(* Logix 5000 project; controller Drives_Line1 1756-L72 rev 20.13; software revision 20.04; part 7 of 21 *)
(* tags used below, declared in another part *)
   Diamtest : BOOL;
   Diamtest_mm : REAL;
   Unwind_1_DiamCalcOn : BOOL;
   Unwinder_2_JEC : REAL;
   Unwinder_2_JLossCrvSpd : REAL[21];
   Unwinder_2_JMaterial : REAL;
   Unwinder_2_LossCrvTrq_Pct : REAL[21];
   Unwinder_2_MatMass : REAL;
   Unwinder_2_MatVolume : REAL;
   Unwinder_2_MaxMass : REAL;
   Unwinder_2_MaxVolume : REAL;
   Unwinder_2_PctPerN : REAL;
   Unwinder_2_RatedTrq : REAL;
   Unwinder_2_RPMPerMPS : REAL;
   zUnwind_2_MaxRate : REAL;
   zUnwind_2_TenRefRate : REAL;
   zUnwind_2_TenSpStall : REAL;
   zUnwind_2_TrqTrimLimMax_Pct : REAL;
   zUnwind_2_TrqTrimLimMin_Pct : REAL;
   zUnwinder_2_JGainQ1Q2 : REAL;
   zUnwinder_2_JGainQ3Q4 : REAL;
   zUnwinder_2_SpdReg_BWMax : REAL;
   zUnwinder_2_SpdReg_BWmin : REAL;
   Bridle_01 : UDT_Bridle_3M;
   EntryConfig : UDT_Config_Zone;
   EntryCtrl : UDT_Control_Zone;
   LineSetpoints : UDT_Setpoints_Line;
   Out_Feedbacks : UDT_Fdbks;
   Out_Status : UDT_Status;
   TestConfig_Unwinder_2 : UDT_Config_Unwinder;
   TestSp_Unwinder_2 : UDT_Setpoints_Unwinder;
   Unwinder_2 : UDT_Unwinder;
   Winder : UDT_Winder;
   zConfigFromMaster : BOOL;
   zPi : REAL;
(* P11_Unwinder_2, continued *)

ROUTINE R09_DiamCalc   (* function block diagram *)
   SHEET 1   // Distance/Angle Integration
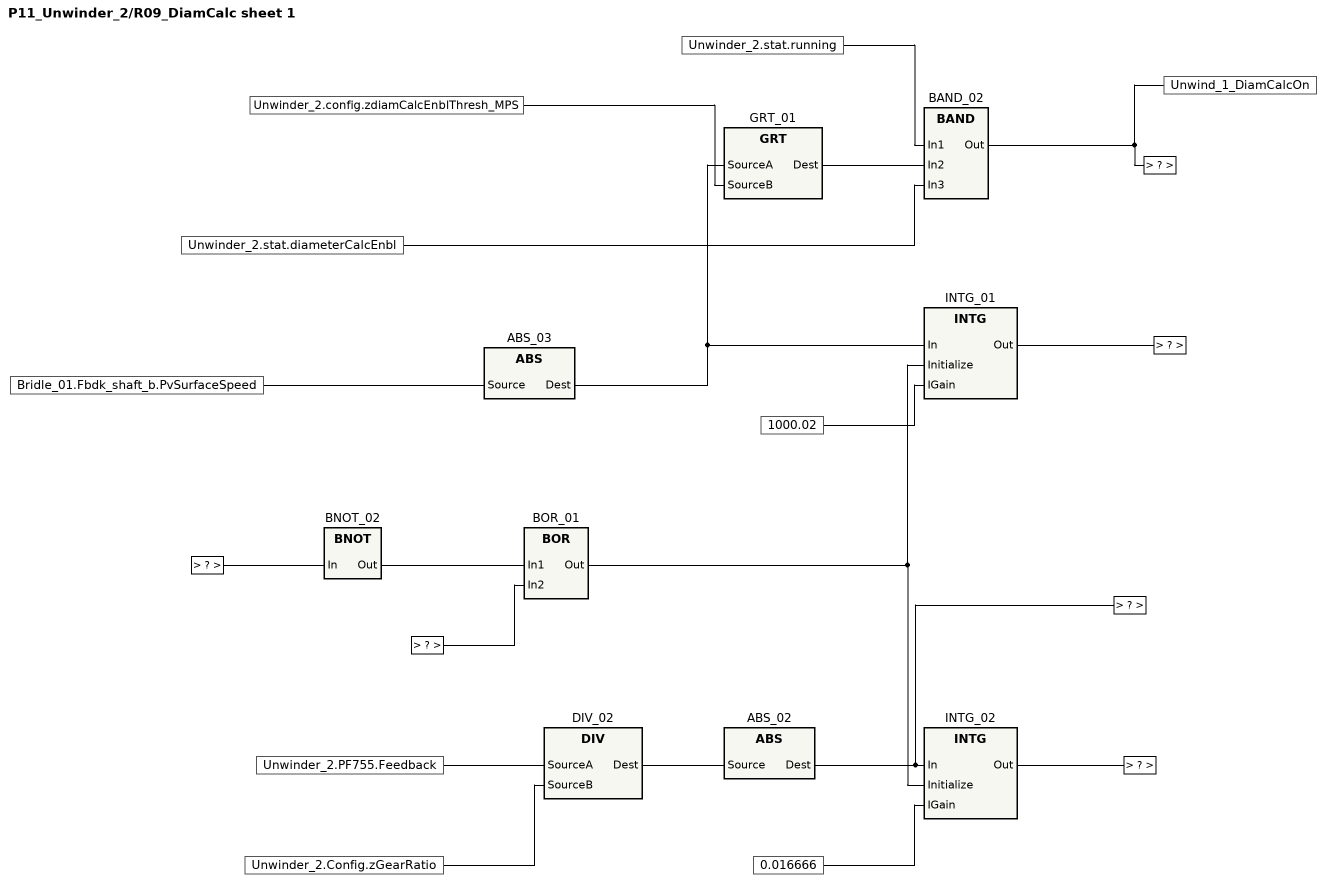
   ABS_03 : ABS(Source := Bridle_01.Fbdk_shaft_b.PvSurfaceSpeed);
   DIV_02 : DIV(SourceA := Unwinder_2.PF755.Feedback, SourceB := Unwinder_2.Config.zGearRatio);
   GRT_01 : GRT(SourceA := ABS_03.Dest, SourceB := Unwinder_2.config.zdiamCalcEnblThresh_MPS);
   ABS_02 : ABS(Source := DIV_02.Dest);
   BAND_02 : BAND(In1 := Unwinder_2.stat.running, In2 := GRT_01.Dest, In3 := Unwinder_2.stat.diameterCalcEnbl);
   WIRE(?) := ABS_02.Dest;
   BNOT_02 : BNOT(In := WIRE(?));
   BOR_01 : BOR(In1 := BNOT_02.Out, In2 := WIRE(?) {feedback});
   INTG_01 : INTG(In := ABS_03.Dest, Initialize := BOR_01.Out, IGain := 1000.02);
   INTG_02 : INTG(In := ABS_02.Dest, Initialize := BOR_01.Out, IGain := 0.016666);
   WIRE(?) := INTG_02.Out;
   WIRE(?) := BAND_02.Out;
   WIRE(?) := INTG_01.Out;
   Unwind_1_DiamCalcOn := BAND_02.Out;
   SHEET 2   // Diameter Calculate
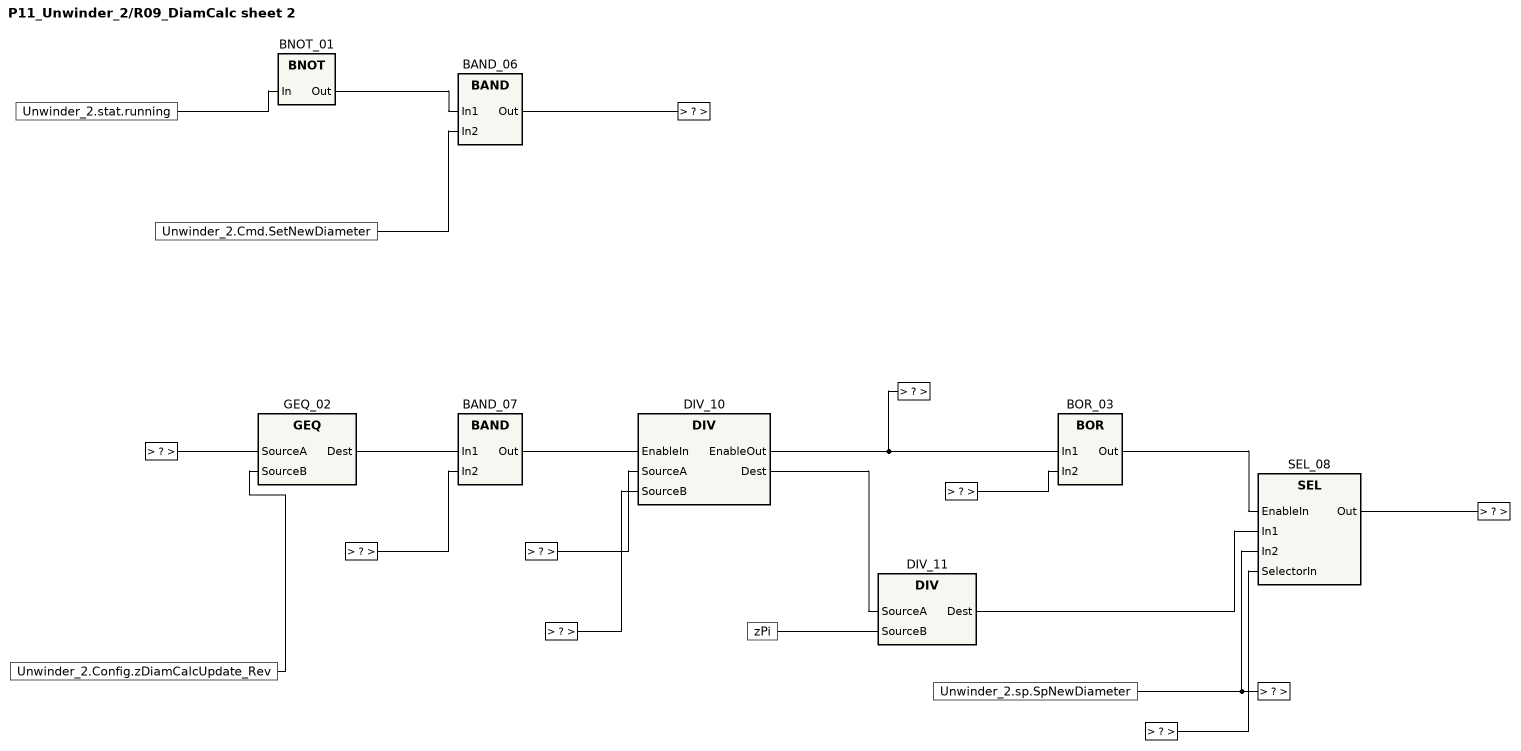
   BNOT_01 : BNOT(In := Unwinder_2.stat.running);
   BAND_06 : BAND(In1 := BNOT_01.Out, In2 := Unwinder_2.Cmd.SetNewDiameter);
   WIRE(?) := BAND_06.Out;
   WIRE(?) := Unwinder_2.sp.SpNewDiameter;
   GEQ_02 : GEQ(SourceA := WIRE(?), SourceB := Unwinder_2.Config.zDiamCalcUpdate_Rev);
   BAND_07 : BAND(In1 := GEQ_02.Dest, In2 := WIRE(?));
   DIV_10 : DIV(EnableIn := BAND_07.Out, SourceA := WIRE(?), SourceB := WIRE(?));
   DIV_11 : DIV(SourceA := DIV_10.Dest, SourceB := zPi);
   WIRE(?) := DIV_10.EnableOut;
   BOR_03 : BOR(In1 := DIV_10.EnableOut, In2 := WIRE(?));
   SEL_08 : SEL(EnableIn := BOR_03.Out, In1 := DIV_11.Dest, In2 := Unwinder_2.sp.SpNewDiameter, SelectorIn := WIRE(?));
   WIRE(?) := SEL_08.Out;
   SHEET 3   // Rate/Magnitude Limit
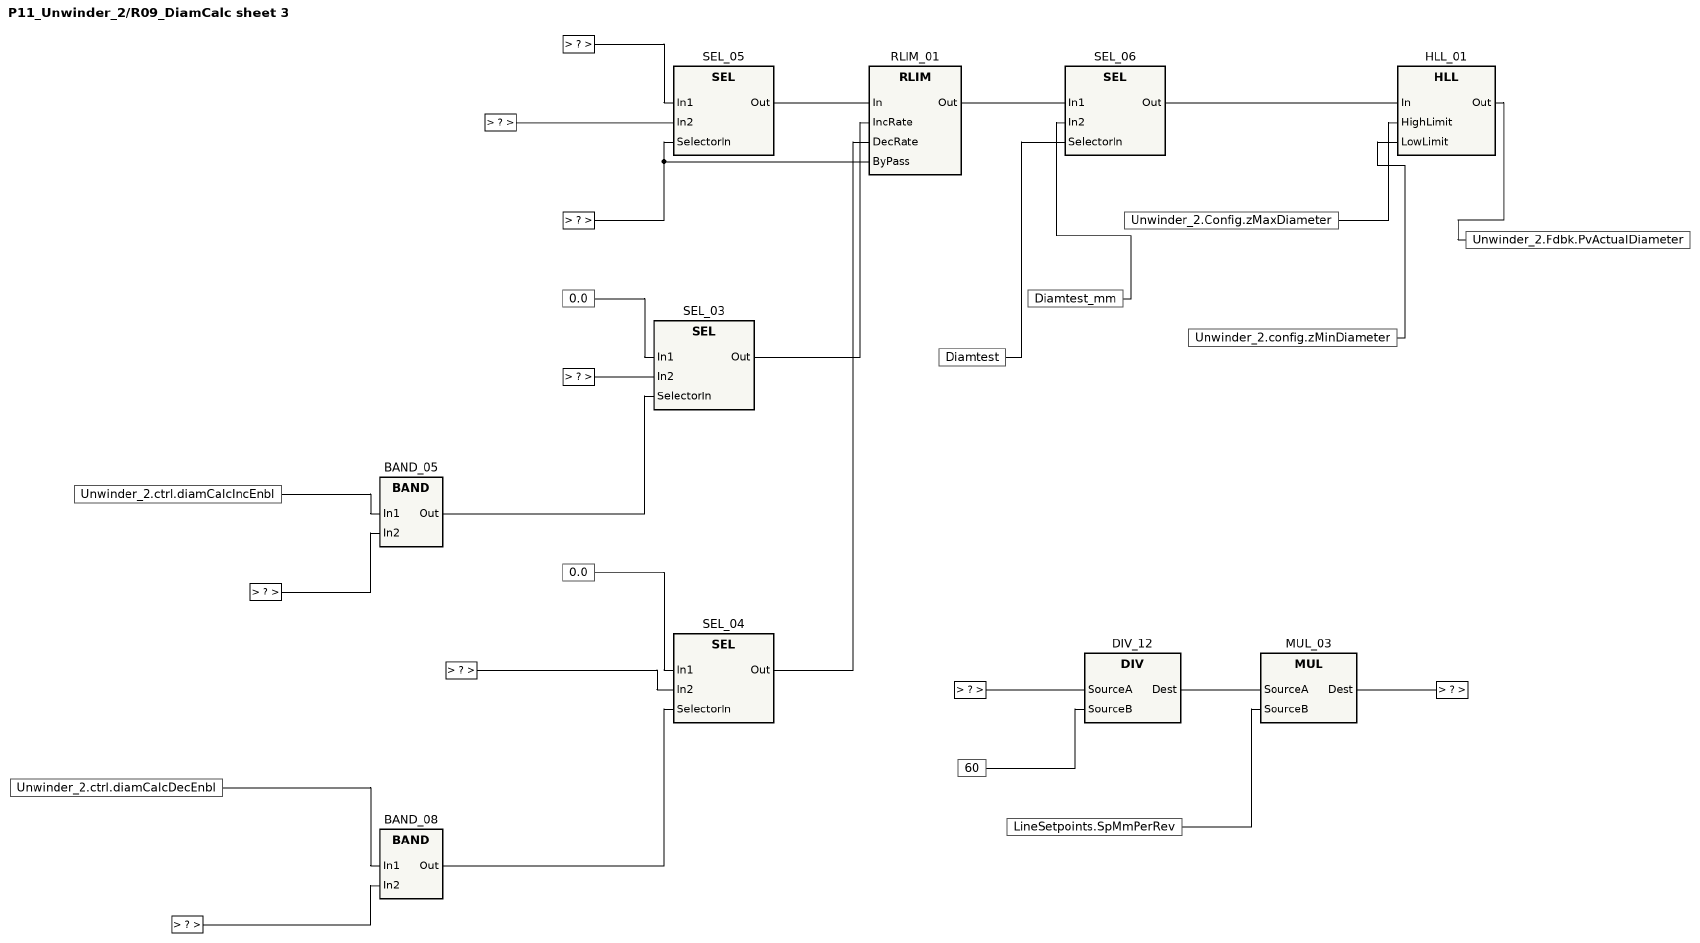
   BAND_08 : BAND(In1 := Unwinder_2.ctrl.diamCalcDecEnbl, In2 := WIRE(?));
   BAND_05 : BAND(In1 := Unwinder_2.ctrl.diamCalcIncEnbl, In2 := WIRE(?));
   SEL_04 : SEL(In1 := 0.0, In2 := WIRE(?), SelectorIn := BAND_08.Out);
   SEL_05 : SEL(In1 := WIRE(?), In2 := WIRE(?), SelectorIn := WIRE(?));
   SEL_03 : SEL(In1 := 0.0, In2 := WIRE(?), SelectorIn := BAND_05.Out);
   RLIM_01 : RLIM(In := SEL_05.Out, IncRate := SEL_03.Out, DecRate := SEL_04.Out, ByPass := WIRE(?));
   SEL_06 : SEL(In1 := RLIM_01.Out, In2 := Diamtest_mm, SelectorIn := Diamtest);
   HLL_01 : HLL(In := SEL_06.Out, HighLimit := Unwinder_2.Config.zMaxDiameter, LowLimit := Unwinder_2.config.zMinDiameter);
   Unwinder_2.Fdbk.PvActualDiameter := HLL_01.Out;
   DIV_12 : DIV(SourceA := WIRE(?), SourceB := 60);
   MUL_03 : MUL(SourceA := DIV_12.Dest, SourceB := LineSetpoints.SpMmPerRev);
   WIRE(?) := MUL_03.Dest;
END_ROUTINE

ROUTINE R10_Calculate   (* structured text *)
   // Calculate
   // Speed Conversion
   //
   // * * * * * * * * * * * * * * * * * * * * * * * * * * *
   //
   // Calculates conversion factor from surface speed [MPS] to rotational speeds [RPM].
   //
   //             Gear Ratio * 1000 [mm/M]
   // RPM/MPS =  -------------------------- * 60
   //             Roll Diameter [mm] * PI
   //
   Unwinder_2_RPMPerMPS := (Unwinder_2.Config.zGearRatio * 1000.0) / (Unwinder_2.Fdbk.PvActualDiameter * zPi) * 60;
   //
   // * * * * * * * * * * * * * * * * * * * * * * * * * * *
   //
   // Calculate
   // (Rated Motor Torque)
   //
   // * * * * * * * * * * * * * * * * * * * * * * * * * * *
   //
   //                       MtrPwrRated [KW] * 9549
   // MtrTrqRated_Nm = ----------------------------
   //                           MtrSpdBase [RPM]
   //
   Unwinder_2_RatedTrq := Unwinder_2.Config.zMotorPwr * 9549 / Unwinder_2.Config.zMtrBaseSpd;
   //
   
   
   //
   // Calculate
   // (Center Winder Inertia)
   //
   // * * * * * * * * * * * * * * * * * * * * * * * * * * *
   //
   // MaterialVolume_m3 = (Pi * (Diam_mm/2000)**2 - Pi * (DiamMinEC_mm/2000)**2) * Width_mm/1000
   //
   Unwinder_2_MatVolume := (zPi * (Unwinder_2.Fdbk.PvActualDiameter/2000)**2)
   - (zPi * (Unwinder_2.Config.zMinDiameter/2000)**2)* (LineSetpoints.WebWidth  / 1000);
   Unwinder_2_MaxVolume:= (zPi * (Unwinder_2.Config.zMaxDiameter/2000)**2)* (LineSetpoints.WebWidth / 1000);
   //
   // MaterialMass_Kg = MaterialVolume_m3 * Density_Kgm3
   //
   Unwinder_2_MatMass := Unwinder_2_MatVolume * LineSetpoints.MaterialDensity ;
   Unwinder_2_MaxMass:= Unwinder_2_MaxVolume * LineSetpoints.MaterialDensity ;
   //
   // JMaterial_Kgm2 = MaterialWeight_Kg / 2 * ((Diam_mm/2000)**2 + (DiamMinEC_mm/2000)**2) / GearRatio**2
   //
   Unwinder_2_JMaterial := Unwinder_2_MatMass / 2 *
   ((Unwinder_2.Fdbk.PvActualDiameter/2000)**2 + (Unwinder_2.Config.zMinDiameter/2000)**2)
    / (Unwinder_2.Config.zGearRatio**2) ;
   //
   // Calculate total reflected inertia [kilogram-meters**2]
   //
   Unwinder_2.Fdbk.PvTotalInertia := Unwinder_2_JEC + Unwinder_2_JMaterial ;
   //
   // * * * * * * * * * * * * * * * * * * * * * * * * * * *
   //
   // Calculate
   // (Normalized Inertia)
   //
   // * * * * * * * * * * * * * * * * * * * * * * * * * * *
   //
   //         J [Kgm**2] * MtrSpdBase [RPM]
   // J_Sec = -------------------------------
   //           9.549 * MtrTrqRated [Nm]
   //
   Unwinder_2.Fdbk.PvNormInertia := (Unwinder_2.Fdbk.PvTotalInertia * Unwinder_2.Config.zMtrBaseSpd)
   / (9.549 * Unwinder_2_RatedTrq) ;
   
   
   (*                         Diam [mm]           100                  1      *)
   (* Conversion_PctPerN =  ----------- * -------------------- * ----------- *)
   (*                         1000 * 2       MtrTrqRated [Nm]      GearRatio  *)
   
   Unwinder_2_PctPerN := Unwinder_2.Fdbk.PvActualDiameter / Unwinder_2.Config.zGearRatio
    / Unwinder_2_RatedTrq / 20.0 ;
   
END_ROUTINE

ROUTINE R11_TenRef   (* function block diagram *)
   SHEET 1   // Tension Reference
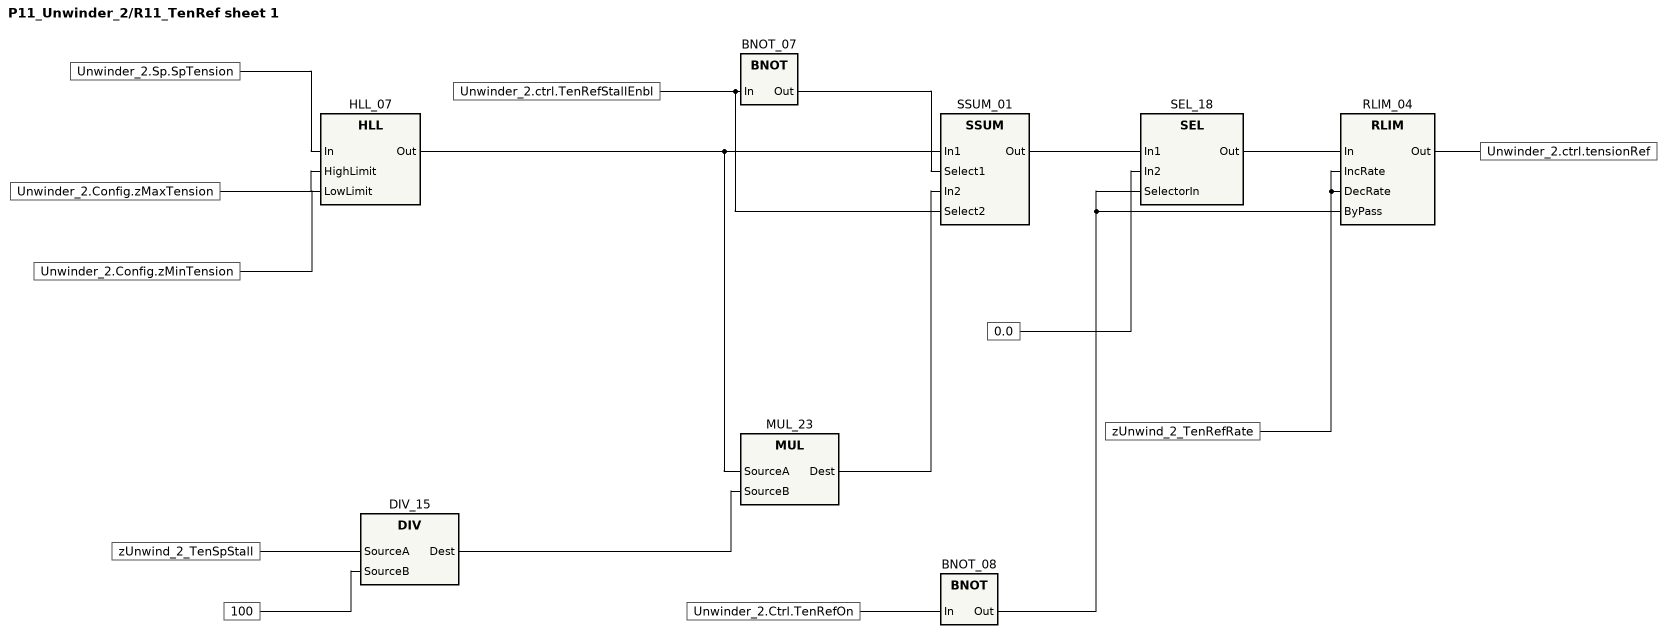
   HLL_07 : HLL(In := Unwinder_2.Sp.SpTension, HighLimit := Unwinder_2.Config.zMaxTension, LowLimit := Unwinder_2.Config.zMinTension);
   DIV_15 : DIV(SourceA := zUnwind_2_TenSpStall, SourceB := 100);
   BNOT_07 : BNOT(In := Unwinder_2.ctrl.TenRefStallEnbl);
   MUL_23 : MUL(SourceA := HLL_07.Out, SourceB := DIV_15.Dest);
   SSUM_01 : SSUM(In1 := HLL_07.Out, Select1 := BNOT_07.Out, In2 := MUL_23.Dest, Select2 := Unwinder_2.ctrl.TenRefStallEnbl);
   BNOT_08 : BNOT(In := Unwinder_2.Ctrl.TenRefOn);
   SEL_18 : SEL(In1 := SSUM_01.Out, In2 := 0.0, SelectorIn := BNOT_08.Out);
   RLIM_04 : RLIM(In := SEL_18.Out, IncRate := zUnwind_2_TenRefRate, DecRate := zUnwind_2_TenRefRate, ByPass := BNOT_08.Out);
   Unwinder_2.ctrl.tensionRef := RLIM_04.Out;
END_ROUTINE

ROUTINE R12_DriveRef   (* function block diagram *)
   SHEET 1   // Speed reference selection
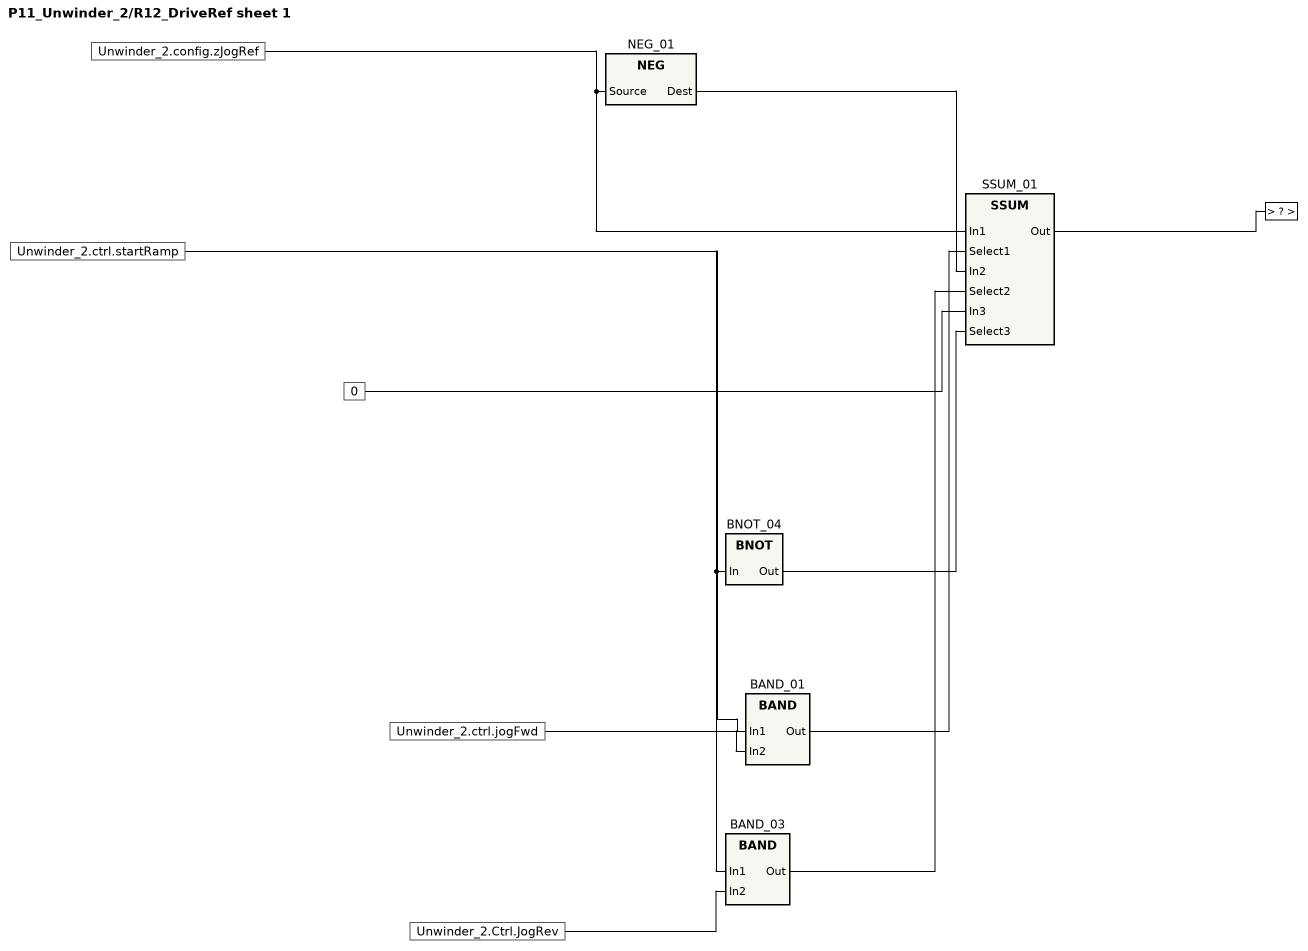
   NEG_01 : NEG(Source := Unwinder_2.config.zJogRef);
   BNOT_04 : BNOT(In := Unwinder_2.ctrl.startRamp);
   BAND_03 : BAND(In1 := Unwinder_2.ctrl.startRamp, In2 := Unwinder_2.Ctrl.JogRev);
   BAND_01 : BAND(In1 := Unwinder_2.ctrl.startRamp, In2 := Unwinder_2.ctrl.jogFwd);
   SSUM_01 : SSUM(In1 := Unwinder_2.config.zJogRef, Select1 := BAND_01.Out, In2 := NEG_01.Dest, Select2 := BAND_03.Out, In3 := 0, Select3 := BNOT_04.Out);
   WIRE(?) := SSUM_01.Out;
   SHEET 2   // S-Curve
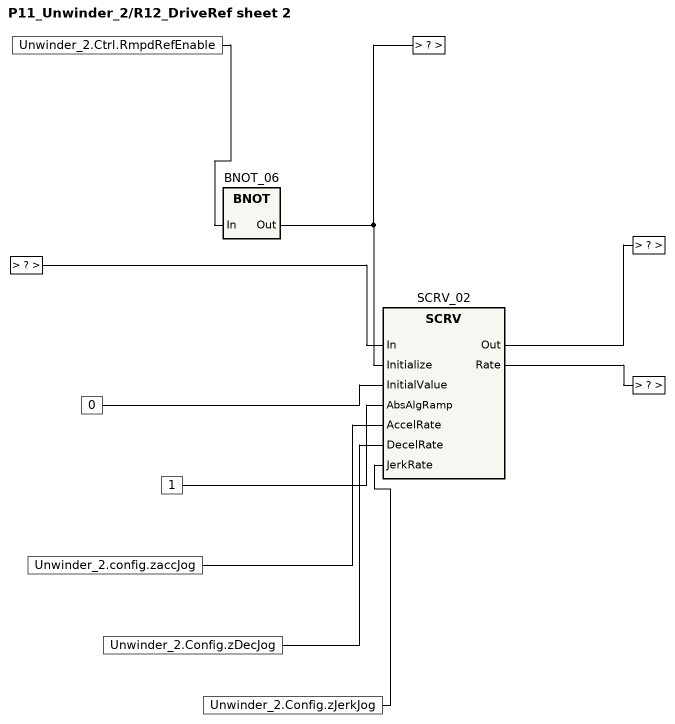
   BNOT_06 : BNOT(In := Unwinder_2.Ctrl.RmpdRefEnable);
   WIRE(?) := BNOT_06.Out;
   SCRV_02 : SCRV(In := WIRE(?), Initialize := BNOT_06.Out, InitialValue := 0, AbsAlgRamp := 1, AccelRate := Unwinder_2.config.zaccJog, DecelRate := Unwinder_2.Config.zDecJog, JerkRate := Unwinder_2.Config.zJerkJog);
   WIRE(?) := SCRV_02.Out;
   WIRE(?) := SCRV_02.Rate;
   SHEET 3   // Select ramped/unramped reference
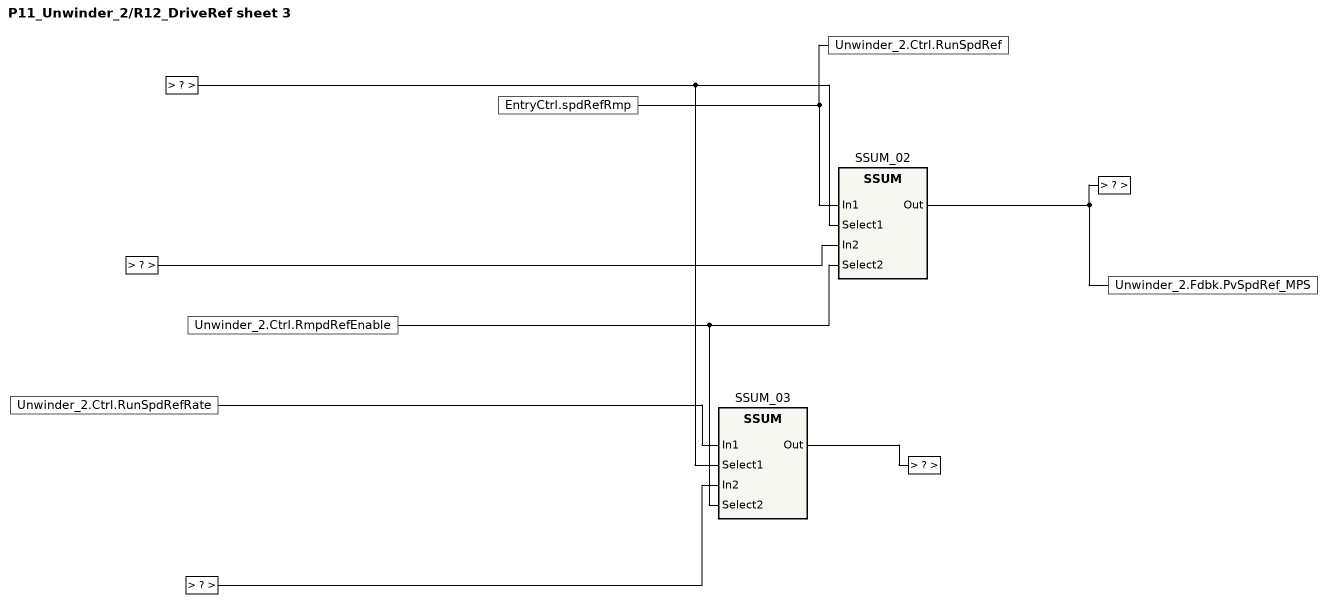
   Unwinder_2.Ctrl.RunSpdRef := EntryCtrl.spdRefRmp;
   SSUM_02 : SSUM(In1 := EntryCtrl.spdRefRmp, Select1 := WIRE(?), In2 := WIRE(?), Select2 := Unwinder_2.Ctrl.RmpdRefEnable);
   WIRE(?) := SSUM_02.Out;
   SSUM_03 : SSUM(In1 := Unwinder_2.Ctrl.RunSpdRefRate, Select1 := WIRE(?), In2 := WIRE(?), Select2 := Unwinder_2.Ctrl.RmpdRefEnable);
   WIRE(?) := SSUM_03.Out;
   Unwinder_2.Fdbk.PvSpdRef_MPS := SSUM_02.Out;
   SHEET 4   // Inertia Compensation
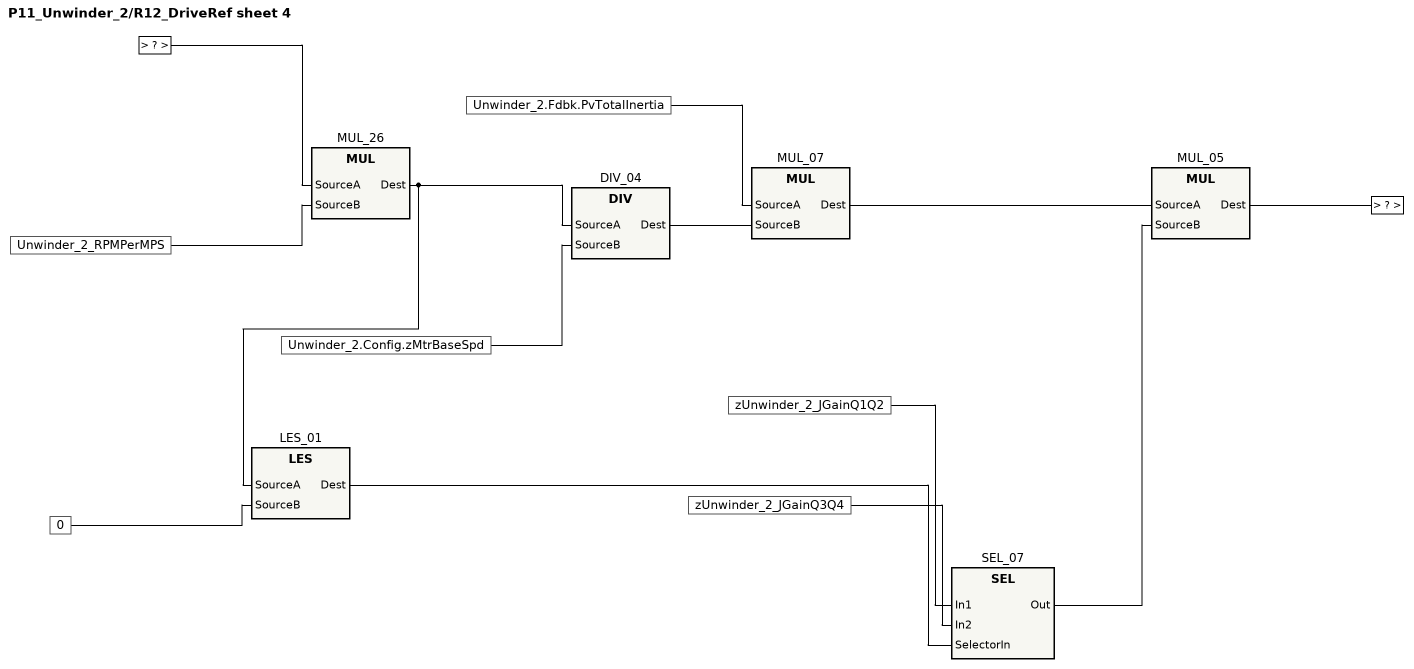
   MUL_26 : MUL(SourceA := WIRE(?), SourceB := Unwinder_2_RPMPerMPS);
   LES_01 : LES(SourceA := MUL_26.Dest, SourceB := 0);
   DIV_04 : DIV(SourceA := MUL_26.Dest, SourceB := Unwinder_2.Config.zMtrBaseSpd);
   MUL_07 : MUL(SourceA := Unwinder_2.Fdbk.PvTotalInertia, SourceB := DIV_04.Dest);
   SEL_07 : SEL(In1 := zUnwinder_2_JGainQ1Q2, In2 := zUnwinder_2_JGainQ3Q4, SelectorIn := LES_01.Dest);
   MUL_05 : MUL(SourceA := MUL_07.Dest, SourceB := SEL_07.Out);
   WIRE(?) := MUL_05.Dest;
   SHEET 5   // Friction and Windage Compensation
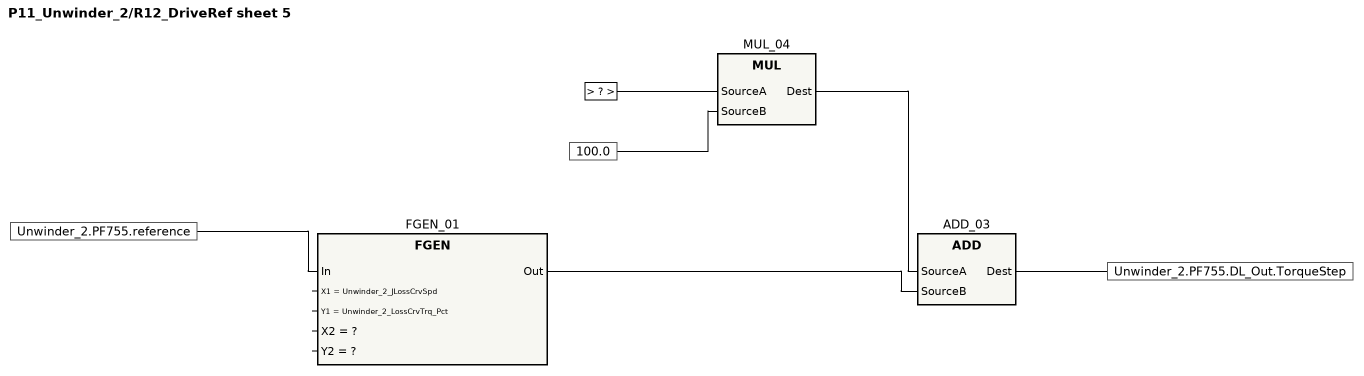
   FGEN_01 : FGEN(In := Unwinder_2.PF755.reference, X1 := Unwinder_2_JLossCrvSpd, Y1 := Unwinder_2_LossCrvTrq_Pct, X2 := ?, Y2 := ?);
   MUL_04 : MUL(SourceA := WIRE(?), SourceB := 100.0);
   ADD_03 : ADD(SourceA := MUL_04.Dest, SourceB := FGEN_01.Out);
   Unwinder_2.PF755.DL_Out.TorqueStep := ADD_03.Dest;
   SHEET 6   // Speed trim
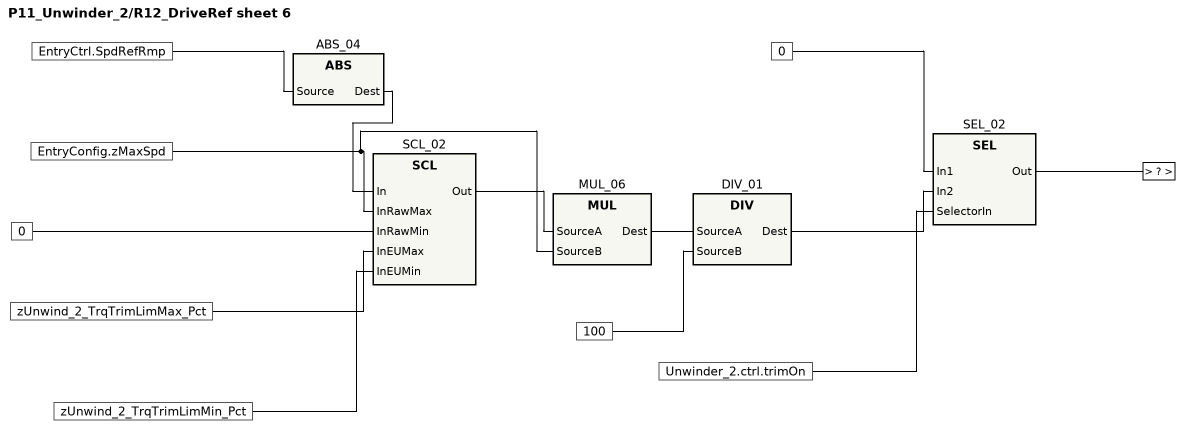
   ABS_04 : ABS(Source := EntryCtrl.SpdRefRmp);
   SCL_02 : SCL(In := ABS_04.Dest, InRawMax := EntryConfig.zMaxSpd, InRawMin := 0, InEUMax := zUnwind_2_TrqTrimLimMax_Pct, InEUMin := zUnwind_2_TrqTrimLimMin_Pct);
   MUL_06 : MUL(SourceA := SCL_02.Out, SourceB := EntryConfig.zMaxSpd);
   DIV_01 : DIV(SourceA := MUL_06.Dest, SourceB := 100);
   SEL_02 : SEL(In1 := 0, In2 := DIV_01.Dest, SelectorIn := Unwinder_2.ctrl.trimOn);
   WIRE(?) := SEL_02.Out;
   SHEET 7   // Final speed reference
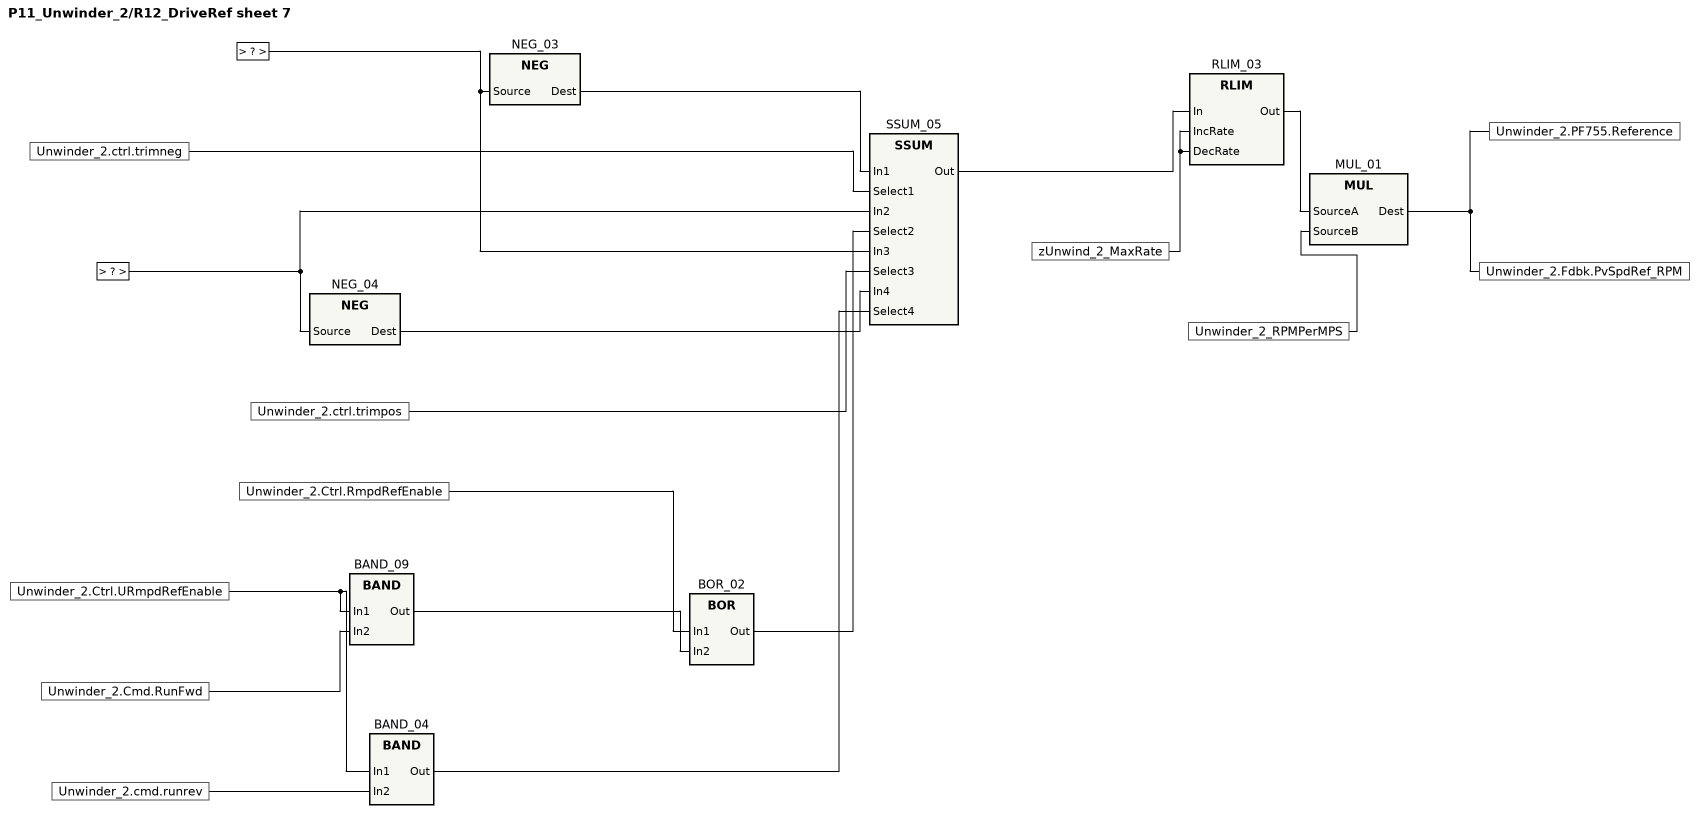
   NEG_04 : NEG(Source := WIRE(?));
   BAND_09 : BAND(In1 := Unwinder_2.Ctrl.URmpdRefEnable, In2 := Unwinder_2.Cmd.RunFwd);
   BAND_04 : BAND(In1 := Unwinder_2.Ctrl.URmpdRefEnable, In2 := Unwinder_2.cmd.runrev);
   NEG_03 : NEG(Source := WIRE(?));
   BOR_02 : BOR(In1 := Unwinder_2.Ctrl.RmpdRefEnable, In2 := BAND_09.Out);
   SSUM_05 : SSUM(In1 := NEG_03.Dest, Select1 := Unwinder_2.ctrl.trimneg, In2 := WIRE(?), Select2 := BOR_02.Out, In3 := WIRE(?), Select3 := Unwinder_2.ctrl.trimpos, In4 := NEG_04.Dest, Select4 := BAND_04.Out);
   RLIM_03 : RLIM(In := SSUM_05.Out, IncRate := zUnwind_2_MaxRate, DecRate := zUnwind_2_MaxRate);
   MUL_01 : MUL(SourceA := RLIM_03.Out, SourceB := Unwinder_2_RPMPerMPS);
   Unwinder_2.Fdbk.PvSpdRef_RPM := MUL_01.Dest;
   Unwinder_2.PF755.Reference := MUL_01.Dest;
   SHEET 8   // Torque reference
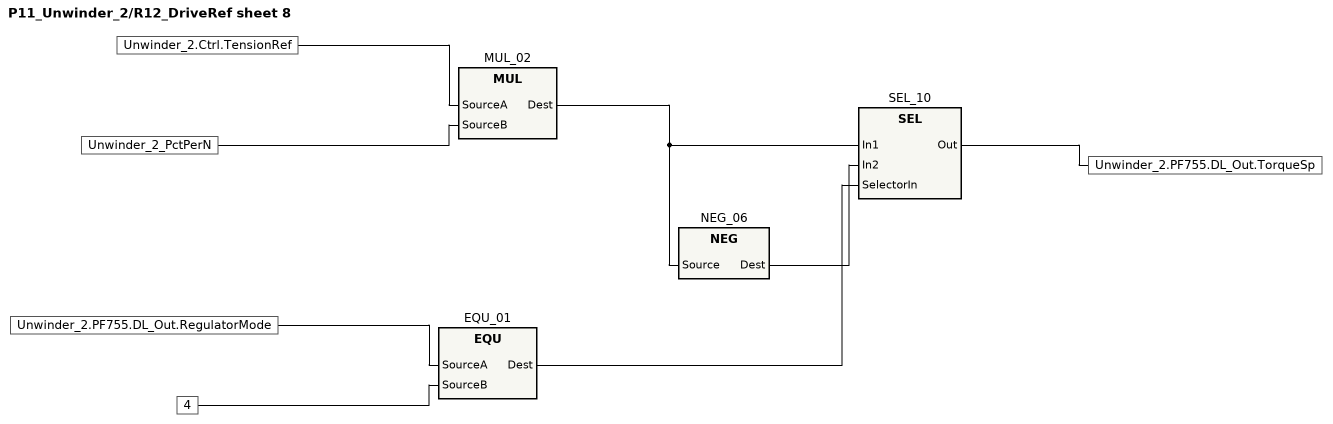
   EQU_01 : EQU(SourceA := Unwinder_2.PF755.DL_Out.RegulatorMode, SourceB := 4);
   MUL_02 : MUL(SourceA := Unwinder_2.Ctrl.TensionRef, SourceB := Unwinder_2_PctPerN);
   NEG_06 : NEG(Source := MUL_02.Dest);
   SEL_10 : SEL(In1 := MUL_02.Dest, In2 := NEG_06.Dest, SelectorIn := EQU_01.Dest);
   Unwinder_2.PF755.DL_Out.TorqueSp := SEL_10.Out;
   SHEET 9   // Speed regulator bandwidth
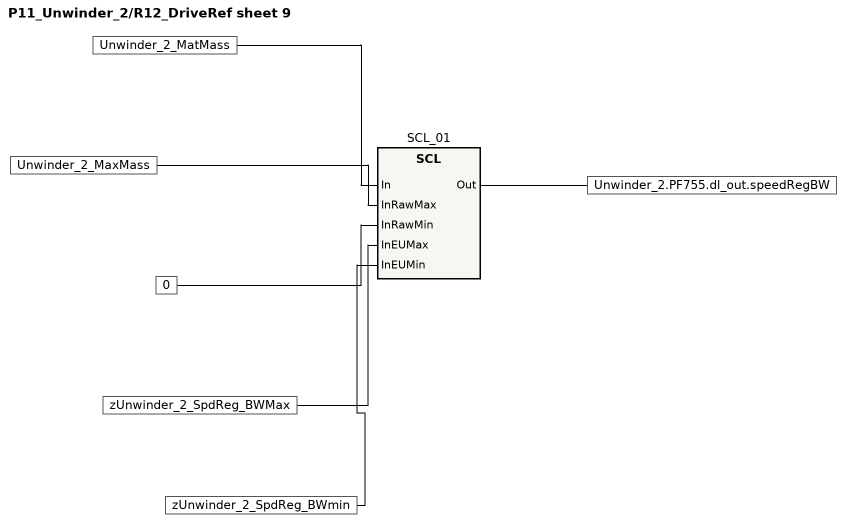
   SCL_01 : SCL(In := Unwinder_2_MatMass, InRawMax := Unwinder_2_MaxMass, InRawMin := 0, InEUMax := zUnwinder_2_SpdReg_BWMax, InEUMin := zUnwinder_2_SpdReg_BWmin);
   Unwinder_2.PF755.dl_out.speedRegBW := SCL_01.Out;
END_ROUTINE

ROUTINE R98_ToDrive   (* ladder *)
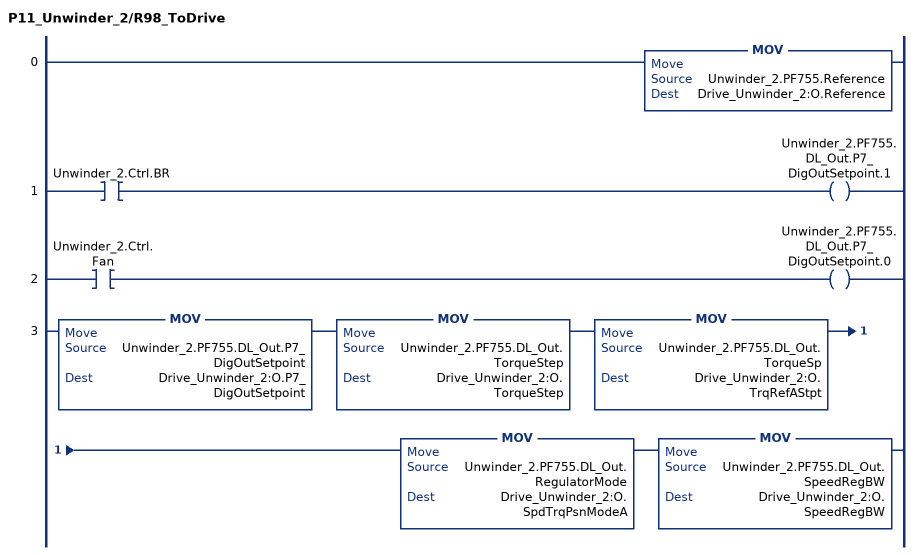
   0: MOV(Unwinder_2.PF755.Reference,Drive_Unwinder_2:O.Reference);
   1: XIC(Unwinder_2.Ctrl.BR)OTE(Unwinder_2.PF755.DL_Out.P7_DigOutSetpoint.1);
   2: XIC(Unwinder_2.Ctrl.Fan)OTE(Unwinder_2.PF755.DL_Out.P7_DigOutSetpoint.0);
   3: MOV(Unwinder_2.PF755.DL_Out.P7_DigOutSetpoint,Drive_Unwinder_2:O.P7_DigOutSetpoint)MOV(Unwinder_2.PF755.DL_Out.TorqueStep,Drive_Unwinder_2:O.TorqueStep)MOV(Unwinder_2.PF755.DL_Out.TorqueSp,Drive_Unwinder_2:O.TrqRefAStpt)MOV(Unwinder_2.PF755.DL_Out.RegulatorMode,Drive_Unwinder_2:O.SpdTrqPsnModeA)MOV(Unwinder_2.PF755.DL_Out.SpeedRegBW,Drive_Unwinder_2:O.SpeedRegBW);
END_ROUTINE

ROUTINE R999_Test   (* ladder *)
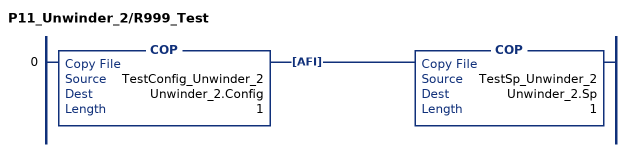
   0: COP(TestConfig_Unwinder_2,Unwinder_2.Config,1)AFI()COP(TestSp_Unwinder_2,Unwinder_2.Sp,1);
END_ROUTINE

ROUTINE R99_To_Master   (* ladder *)
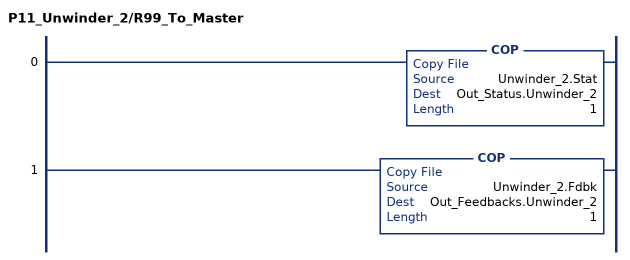
   0: COP(Unwinder_2.Stat,Out_Status.Unwinder_2,1);
   1: COP(Unwinder_2.Fdbk,Out_Feedbacks.Unwinder_2,1);
END_ROUTINE
END_PROGRAM

PROGRAM P12_Pinchroll_1   (* main routine R00_Main *)
VAR
   ABS_01 : FBD_MATH_ADVANCED;
   BAND_01 : FBD_BOOLEAN_AND := (In1 := 1, In3 := 1, In4 := 1, In5 := 1, In6 := 1, In7 := 1, In8 := 1);
   BAND_02 : FBD_BOOLEAN_AND := (In3 := 1, In4 := 1, In5 := 1, In6 := 1, In7 := 1, In8 := 1);
   BAND_03 : FBD_BOOLEAN_AND := (In3 := 1, In4 := 1, In5 := 1, In6 := 1, In7 := 1, In8 := 1);
   BAND_04 : FBD_BOOLEAN_AND := (In3 := 1, In4 := 1, In5 := 1, In6 := 1, In7 := 1, In8 := 1);
   BNOT_01 : FBD_BOOLEAN_NOT := (Out := 1);
   BOR_01 : FBD_BOOLEAN_OR;
   IO_State_Pinch_1 : INT := 4;
   IO_State_Tmp_Pinch_1 : INT := 16384;
   LES_01 : FBD_COMPARE := (SourceB := 0.016, Dest := 1);
   MUL_01 : FBD_MATH := (SourceB := 1283.6122);
   Pinchroll_1_RPMPerMPS : REAL := 1283.6122;
   RLIM_01 : RATE_LIMITER := (IncRate := 0.1, DecRate := 0.1, RTSTime := 1, DeltaT := 0.05);
   SSUM_01 : SELECTED_SUMMER := (Gain1 := 1.0, Gain2 := 1.0, Gain3 := 1.0, Gain4 := 1.0, Select4 := 1, Gain5 := 1.0, Gain6 := 1.0, Gain7 := 1.0, Gain8 := 1.0);
   SUB_01 : FBD_MATH;
   TofReset : TIMER := (PRE := 1000, ACC := 1000);
   TonNoResponse : TIMER := (PRE := 2500);
END_VAR

ROUTINE R00_Main   (* ladder *)
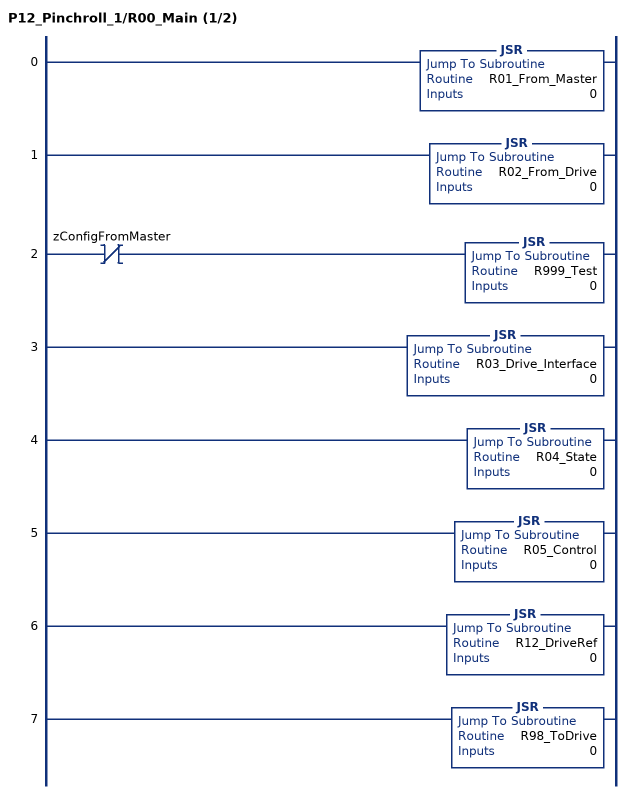
   0: JSR(R01_From_Master,0);
   1: JSR(R02_From_Drive,0);
   2: XIO(zConfigFromMaster)JSR(R999_Test,0);
   3: JSR(R03_Drive_Interface,0);
   4: JSR(R04_State,0);
   5: JSR(R05_Control,0);
   6: JSR(R12_DriveRef,0);
   7: JSR(R98_ToDrive,0);
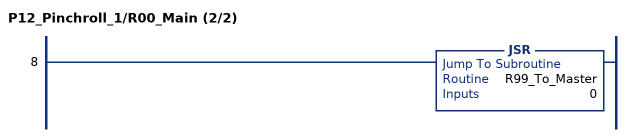
   8: JSR(R99_To_Master,0);
END_ROUTINE
